FUNCTION_BLOCK UintComparator IMPLEMENTS I_Comparator,I_StepCondition
VAR_INPUT
END_VAR
VAR_OUTPUT
END_VAR
VAR
	uiSelector 		: UINT;
	rInternTarget1 	: REFERENCE TO UINT;
	rInternTarget2 	: REFERENCE TO UINT;
	bValue			: BOOL;
END_VAR

IF NOT __ISVALIDREF( rInternTarget1 )
OR NOT __ISVALIDREF( rInternTarget1 )
THEN
	uiSelector := 0;
END_IF 

CASE uiSelector OF

	0:;
		
	10:
		bValue := mEquals(rInternTarget1,rInternTarget2);
		
	20:
		bValue := mGreaterThan(rInternTarget1,rInternTarget2);
	
	30:
		bValue := mLessThan(rInternTarget1,rInternTarget2);
	
	40:
		bValue := mGreaterEquals(rInternTarget1,rInternTarget2);
		
	50:
		bValue := mLessEquals(rInternTarget1,rInternTarget2);
		
END_CASE


PROPERTY getValue : BOOL
GET
getValue := bValue;
END_GET
END_PROPERTY

METHOD mEquals : BOOL;
VAR_INPUT
	rTarget1 : REFERENCE TO UINT;
	rTarget2 : REFERENCE TO UINT;
END_VAR
uiSelector := 10;
rInternTarget1 REF= rTarget1;
rInternTarget2 REF= rTarget2;

mEquals := ( rTarget1 = rTarget2 );
END_METHOD

METHOD PUBLIC mGreaterEquals : BOOL
VAR_INPUT
	rTarget1 : REFERENCE TO UINT;
	rTarget2 : REFERENCE TO UINT;
END_VAR
uiSelector := 40;
rInternTarget1 REF= rTarget1;
rInternTarget2 REF= rTarget2;

mGreaterEquals := ( rTarget1 >= rTarget2 );
END_METHOD

METHOD mGreaterThan : BOOL;
VAR_INPUT
	rTarget1 : REFERENCE TO UINT;
	rTarget2 : REFERENCE TO UINT;
END_VAR
uiSelector := 20;
rInternTarget1 REF= rTarget1;
rInternTarget2 REF= rTarget2;

mGreaterThan := ( rTarget1 >= rTarget2 );
END_METHOD

METHOD mLessEquals : BOOL
VAR_INPUT
	rTarget1 : REFERENCE TO UINT;
	rTarget2 : REFERENCE TO UINT;
END_VAR
uiSelector := 50;
rInternTarget1 REF= rTarget1;
rInternTarget2 REF= rTarget2;

mLessEquals := ( rTarget1 <= rTarget2 );
END_METHOD

METHOD mLessThan : BOOL;
VAR_INPUT
	rTarget1 : REFERENCE TO UINT;
	rTarget2 : REFERENCE TO UINT;
END_VAR
uiSelector := 30;
rInternTarget1 REF= rTarget1;
rInternTarget2 REF= rTarget2;

mLessThan := ( rTarget1 < rTarget2 );
END_METHOD


PROPERTY setValue : BOOL
SET
bValue := setValue;
END_SET
END_PROPERTY

END_FUNCTION_BLOCK

(* stored: Version 1.1.0.1, ProductVersion 3.1.4024.0
   POU UintComparator: Id {c3538391-8178-426b-8224-2c8c8631c8cc}, SpecialFunc None
   Property getValue: Id {b035f5c0-b3d9-4e77-b7e0-2d7e9fc6953c}
   Get Get: Id {bbb91f6a-1d65-496c-99a4-e5223dff608b}
   Method mEquals: Id {9dfb4363-47be-4e33-bb70-454ad60c93e8}
   Method mGreaterEquals: Id {7e4c987c-fe00-48c4-9cf5-8c637cbfeefe}
   Method mGreaterThan: Id {91d34b43-fc7c-44fe-a6d9-a896f1425185}
   Method mLessEquals: Id {2bd9425f-805a-45a5-8f1d-134f0d8c116a}
   Method mLessThan: Id {0b685c53-bb9a-4f2a-870d-f38717898207}
   Property setValue: Id {6c9d6573-9f69-4bf2-84c3-df921f23e5eb}
   Set Set: Id {8e52679c-e344-4394-a23c-1197e935ed4f} *)
